// TIA Portal V16 export
// export: Created 2022-11-17T11:55:24.7540056Z, ExportSetting WithDefaults, DisplayName Totally Integrated Automation Portal, DisplayVersion V16 Update 6, DisplayName TIA Portal Version Control Interface, DisplayVersion V16 Update 2, DisplayName TIA Portal Openness, DisplayVersion V16 Update 6, DisplayName SINAMICS Startdrive Advanced, DisplayVersion V16 Update 5, DisplayName SINAMICS Startdrive G130, G150, S120, S150, SINAMICS MV, S210, DisplayVersion V16 Update 5, DisplayName SINAMICS Startdrive G110M, G120, G120C, G120D, G120P, G115D, DisplayVersion V16 Update 5, DisplayName STEP 7 Professional, DisplayVersion V16 Update 6, DisplayName STEP 7 Safety, DisplayVersion V16, DisplayName WinCC Advanced, DisplayVersion V16 Update 6
DATA_BLOCK "DB01_Osr"   // DB1
{ S7_Optimized_Access := 'FALSE' }
AUTHOR : Robopac
VERSION : 0.0
// stored: AutoNumber false, IsOnlyStoredInLoadMemory false, IsWriteProtectedInAS false
   VAR RETAIN
      osr1 : Bool := TRUE;   // Used
      osr2 : Bool := FALSE;   // Used
      osr3 : Bool := FALSE;   // Used
      osr4 : Bool := FALSE;   // Used
      osr5 : Bool := FALSE;   // Used
      osr6 : Bool := TRUE;   // Used
      osr7 : Bool := TRUE;   // Used
      osr8 : Bool := FALSE;   // Used
      osr9 : Bool := TRUE;   // Used
      osr10 : Bool := FALSE;   // Used
      osr11 : Bool := FALSE;   // Used
      osr12 : Bool := FALSE;   // Used
      osr13 : Bool := FALSE;   // Used
      osr14 : Bool := FALSE;   // Used
      osr15 : Bool := TRUE;   // Used
      osr16 : Bool := FALSE;   // Used
      osr17 : Bool := TRUE;   // Used
      osr18 : Bool := TRUE;   // Used
      osr19 : Bool := TRUE;   // Used
      osr20 : Bool := TRUE;   // Used
      osr21 : Bool := TRUE;   // Used
      osr22 : Bool := TRUE;   // Used
      osr23 : Bool := FALSE;   // Used
      osr24 : Bool := FALSE;   // Used
      osr25 : Bool := FALSE;   // Used
      osr26 : Bool := FALSE;   // Used
      osr27 : Bool := FALSE;   // Used
      osr28 : Bool := FALSE;   // Used
      osr29 : Bool := FALSE;   // Used
      osr30 : Bool := TRUE;   // Used
      osr31 : Bool := TRUE;   // Used
      osr32 : Bool := TRUE;   // Used
      osr33 : Bool := TRUE;   // Used
      osr34 : Bool := TRUE;   // Used
      osr35 : Bool := FALSE;   // Used
      osr36 : Bool := FALSE;   // Used
      osr37 : Bool := TRUE;
      osr38 : Bool := FALSE;   // Used
      osr39 : Bool := TRUE;   // Used
      osr40 : Bool := FALSE;   // Used
      osr41 : Bool := TRUE;   // Used
      osr42 : Bool := TRUE;
      osr43 : Bool := TRUE;
      osr44 : Bool := FALSE;
      osr45 : Bool := FALSE;   // Used
      osr46 : Bool := FALSE;   // Used
      osr47 : Bool := FALSE;
      osr48 : Bool := FALSE;
      osr49 : Bool := FALSE;
      osr50 : Bool := TRUE;
      osr51 : Bool := FALSE;
      osr52 : Bool := TRUE;
      osr53 : Bool := FALSE;
      osr54 : Bool := FALSE;
      osr55 : Bool := FALSE;
      osr56 : Bool := TRUE;
      osr57 : Bool := FALSE;
      osr58 : Bool := FALSE;
      osr59 : Bool := FALSE;
      osr60 : Bool := TRUE;
      osr61 : Bool := FALSE;
      osr62 : Bool := FALSE;
      osr63 : Bool := FALSE;
      osr64 : Bool := FALSE;
      osr65 : Bool := FALSE;
      osr66 : Bool := FALSE;
      osr67 : Bool := TRUE;
      osr68 : Bool := FALSE;
      osr69 : Bool := TRUE;
      osr70 : Bool := FALSE;
      osr71 : Bool := FALSE;
      osr72 : Bool := FALSE;
      osr73 : Bool := FALSE;
      osr74 : Bool := TRUE;
      osr75 : Bool := TRUE;
      osr76 : Bool := FALSE;
      osr77 : Bool := TRUE;
      osr78 : Bool := TRUE;
      osr79 : Bool := FALSE;
      osr80 : Bool := FALSE;
      osr81 : Bool := FALSE;   // Used
      osr82 : Bool := FALSE;   // Used
      osr83 : Bool := FALSE;
      osr84 : Bool := FALSE;
      osr85 : Bool := FALSE;
      osr86 : Bool := FALSE;
      osr87 : Bool := FALSE;
      osr88 : Bool := TRUE;
      osr89 : Bool := FALSE;
      osr90 : Bool := FALSE;   // Used
      osr91 : Bool := FALSE;
      osr92 : Bool := FALSE;
      osr93 : Bool := TRUE;
      osr94 : Bool := TRUE;
      osr95 : Bool := TRUE;
      osr96 : Bool := TRUE;
   END_VAR
BEGIN
END_DATA_BLOCK
